// TIA Portal V16 export
// export: Created 2022-07-21T09:35:30.9300272Z, ExportSetting WithDefaults, DisplayName Totally Integrated Automation Portal, DisplayVersion V16 Update 4, DisplayName TIA Portal Version Control Interface, DisplayVersion V16 Update 2, DisplayName TIA Portal Openness, DisplayVersion V16 Update 4, DisplayName SINAMICS Startdrive Advanced, DisplayVersion V16 Update 5, DisplayName SINAMICS Startdrive G130, G150, S120, S150, SINAMICS MV, S210, DisplayVersion V16 Update 5, DisplayName SINAMICS Startdrive G110M, G120, G120C, G120D, G120P, G115D, DisplayVersion V16 Update 5, DisplayName STEP 7 Professional, DisplayVersion V16 Update 4, DisplayName STEP 7 Safety, DisplayVersion V16, DisplayName WinCC Advanced, DisplayVersion V16 Update 4
FUNCTION_BLOCK "fbTransport"   // FB34, LAD
TITLE = Transport handling / Obsługa transportu
{ S7_Optimized_Access := 'TRUE' }
VERSION : 0.1
// stored: AutoNumber true, IsIECCheckEnabled false, IsRetainMemResEnabled false, MemoryReserve 100, SetENOAutomatically false, UDAEnableTagReadback false
   VAR_INPUT
      inEnable { ExternalAccessible := 'False'; ExternalVisible := 'False'; ExternalWritable := 'False'} : Bool;   // Ogólne zezwolenie / General release
      inStartRelease { ExternalAccessible := 'False'; ExternalVisible := 'False'; ExternalWritable := 'False'} : Bool;   // Warunki na rozpoczęcie transportu / Conditions to start transport
      inLogOn { ExternalAccessible := 'False'; ExternalVisible := 'False'; ExternalWritable := 'False'} : Bool;   // Sygnał rozpoczynający transport / Start transport
      inLogOff { ExternalAccessible := 'False'; ExternalVisible := 'False'; ExternalWritable := 'False'} : Bool;   // Warunki na zakończenie transportu / Conditions to end transport
      inCancelTransport { ExternalAccessible := 'False'; ExternalVisible := 'False'; ExternalWritable := 'False'} : Bool;   // Natychmiastowe zakończenie transportu / Immediate end transport
      inNextPrevScan { ExternalAccessible := 'False'; ExternalVisible := 'False'; ExternalWritable := 'False'} : USInt;   // Dystans kolejnego przenośnika / Another conveyor distance
      inNextOnSpeed { ExternalAccessible := 'False'; ExternalVisible := 'False'; ExternalWritable := 'False'} : Bool;   // Następny przenośnik jedzie z nominalną prędkością / Next conveyor move with normal speed
      inHeadToHead { ExternalAccessible := 'False'; ExternalVisible := 'False'; ExternalWritable := 'False'} : UInt;   // Dystans czoło obiektu do czoła następnego / Distance head to next head
      inMinusToleranceHeadToHead { ExternalAccessible := 'False'; ExternalVisible := 'False'; ExternalWritable := 'False'} : UInt;   // Toleracja dystansu H2H / Distance tolerance H2H
      inTailToHead { ExternalAccessible := 'False'; ExternalVisible := 'False'; ExternalWritable := 'False'} : UInt;   // Dystans tył obiektu do następnego czoła / Distance tail to next head
      inMinusToleranceTailToHead { ExternalAccessible := 'False'; ExternalVisible := 'False'; ExternalWritable := 'False'} : UInt;   // Tolerancja dystansu T2H / Distance tolerance T2H
      inHeadToHeadTillCancel { ExternalAccessible := 'False'; ExternalVisible := 'False'; ExternalWritable := 'False'} : UInt := 0;   // Dystans do warunkowego zakończenia transportu / Distance to conditional end transport
   END_VAR
   VAR_IN_OUT
      ioData : "typeConveyor";   // Struktura conveyor / Conveyor structure
   END_VAR
   VAR
      sInternalEnable { ExternalAccessible := 'False'; ExternalVisible := 'False'; ExternalWritable := 'False'} : Bool;
   END_VAR
   VAR RETAIN
      sCounterHeadToHead { ExternalAccessible := 'False'; ExternalVisible := 'False'; ExternalWritable := 'False'} : UInt;
      sCounterTailToHead { ExternalAccessible := 'False'; ExternalVisible := 'False'; ExternalWritable := 'False'} : UInt;
      sCounterHeadToLogOn { ExternalAccessible := 'False'; ExternalVisible := 'False'; ExternalWritable := 'False'} : UInt;
      sMemRELogOn { ExternalAccessible := 'False'; ExternalVisible := 'False'; ExternalWritable := 'False'} : Bool;
      sMemRETransport { ExternalAccessible := 'False'; ExternalVisible := 'False'; ExternalWritable := 'False'} : Bool;
      sMemFETransport { ExternalAccessible := 'False'; ExternalVisible := 'False'; ExternalWritable := 'False'} : Bool;
   END_VAR
   VAR
      sHeadToHeadCancel : Bool;
   END_VAR
   VAR_TEMP
      tDistancePrevScan : USInt;
      tReqHeadToHead : UInt;
      tReqTailToHead : UInt;
      tTransportReady : Bool;
      tEndTransport : Bool;
      tDistanceReached : Bool;
      tReqMinusToleranceHeadToHead : UInt;
      tReqMinusToleranceTailToHead : UInt;
      tReset : Bool;
   END_VAR
   VAR_TEMP   // added for the SCL form of the ladder/FBD networks
      _w1 : Bool;
   END_VAR
BEGIN

REGION Network 1: Enable / Zezwolenie
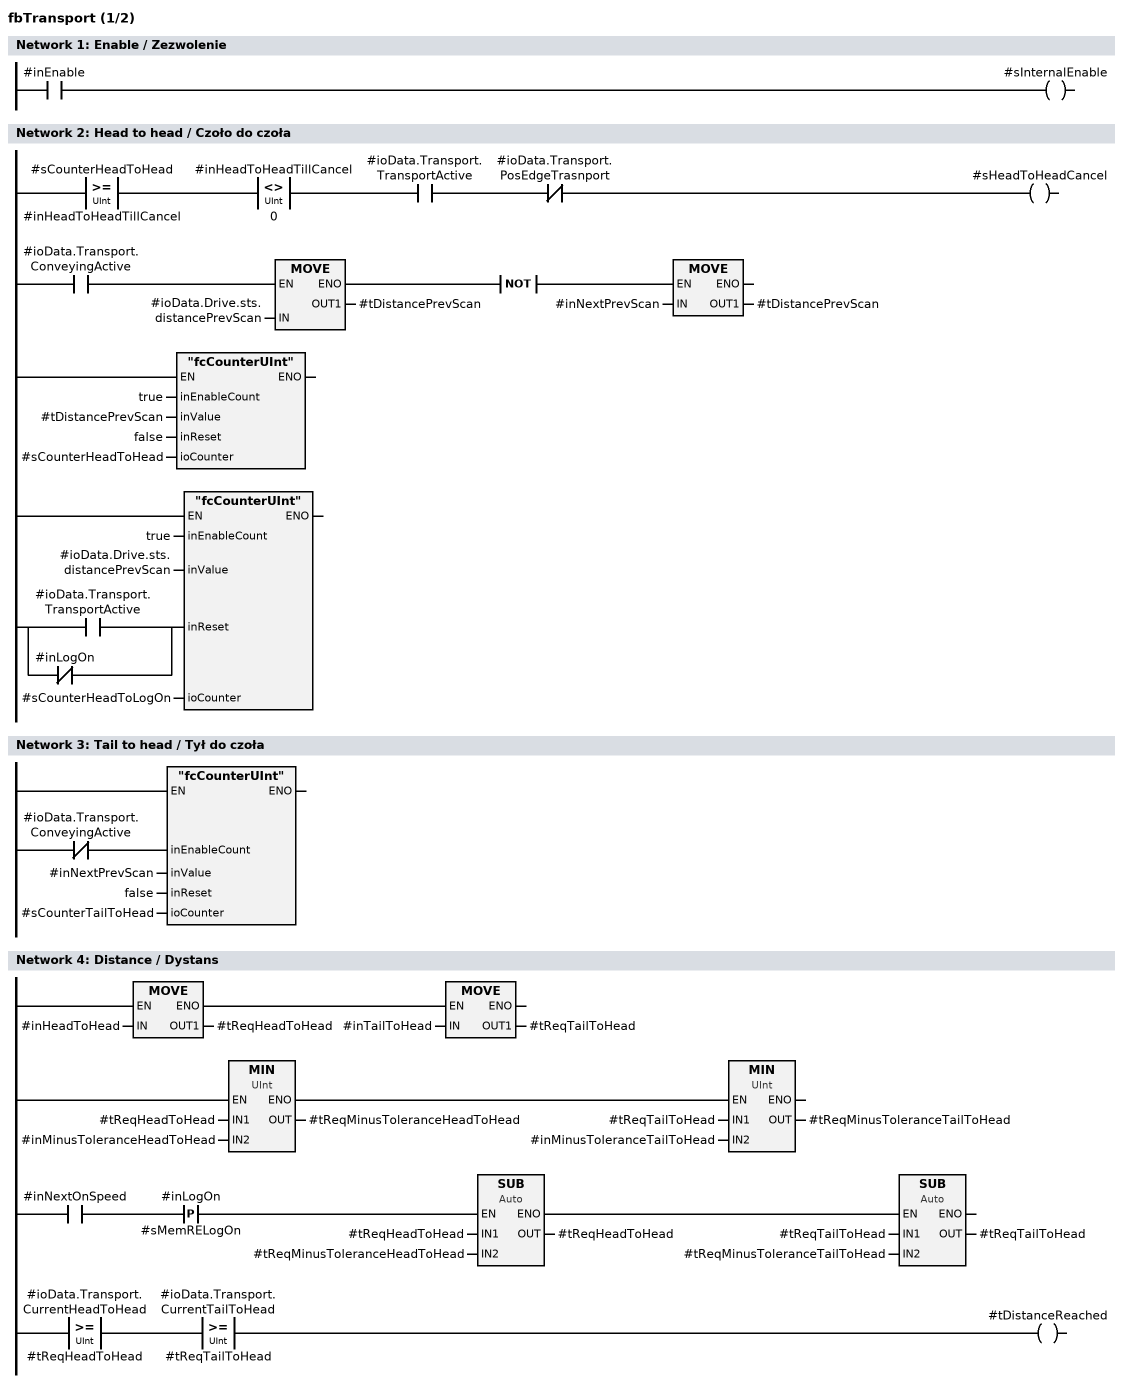
   RUNG wire#powerrail
      Contact( #inEnable )
      Coil( #sInternalEnable )
   END_RUNG
   // the same network as SCL:
   #sInternalEnable := #inEnable;
END_REGION

REGION Network 2: Head to head / Czoło do czoła
   RUNG wire#powerrail
      { S7_Templates := "SrcType := UInt" } GE_Contact(in1 := #sCounterHeadToHead, in2 := #inHeadToHeadTillCancel)
      { S7_Templates := "SrcType := UInt" } NE_Contact(in1 := #inHeadToHeadTillCancel, in2 := 0)
      Contact( #ioData.Transport.TransportActive )
      I_Contact( #ioData.Transport.PosEdgeTrasnport )
      Coil( #sHeadToHeadCancel )
   END_RUNG
   RUNG wire#powerrail
      Contact( #ioData.Transport.ConveyingActive )
      Move(in := #ioData.Drive.sts.distancePrevScan, out1 => #tDistancePrevScan)
      Not()
      Move(in := #inNextPrevScan, out1 => #tDistancePrevScan)
   END_RUNG
   RUNG wire#powerrail
      "fcCounterUInt"(inEnableCount := true, inValue := #tDistancePrevScan, inReset := false, ioCounter := #sCounterHeadToHead)
   END_RUNG
   RUNG wire#powerrail
      "fcCounterUInt"(inReset := wire#w1, inEnableCount := true, inValue := #ioData.Drive.sts.distancePrevScan, ioCounter := #sCounterHeadToLogOn)
   END_RUNG
   RUNG wire#powerrail
      Contact( #ioData.Transport.TransportActive )
   END_RUNG wire#w1
   RUNG wire#powerrail
      I_Contact( #inLogOn )
   END_RUNG wire#w1
   // the same network as SCL:
   #sHeadToHeadCancel := (#sCounterHeadToHead >= #inHeadToHeadTillCancel) AND (#inHeadToHeadTillCancel <> 0) AND #ioData.Transport.TransportActive AND NOT #ioData.Transport.PosEdgeTrasnport;
   IF #ioData.Transport.ConveyingActive THEN
       #tDistancePrevScan := #ioData.Drive.sts.distancePrevScan;
   END_IF;
   IF NOT #ioData.Transport.ConveyingActive THEN #tDistancePrevScan := #inNextPrevScan; END_IF;
   "fcCounterUInt"(inEnableCount := true,
                   inValue := #tDistancePrevScan,
                   inReset := false,
                   ioCounter := #sCounterHeadToHead);
   "fcCounterUInt"(inEnableCount := true,
                   inValue := #ioData.Drive.sts.distancePrevScan,
                   inReset := #ioData.Transport.TransportActive OR NOT #inLogOn,
                   ioCounter := #sCounterHeadToLogOn);
END_REGION

REGION Network 3: Tail to head / Tył do czoła
   RUNG wire#powerrail
      "fcCounterUInt"(inEnableCount := wire#w1, inValue := #inNextPrevScan, inReset := false, ioCounter := #sCounterTailToHead)
   END_RUNG
   RUNG wire#powerrail
      I_Contact( #ioData.Transport.ConveyingActive )
   END_RUNG wire#w1
   // the same network as SCL:
   "fcCounterUInt"(inEnableCount := NOT #ioData.Transport.ConveyingActive,
                   inValue := #inNextPrevScan,
                   inReset := false,
                   ioCounter := #sCounterTailToHead);
END_REGION

REGION Network 4: Distance / Dystans
   RUNG wire#powerrail
      Move(in := #inHeadToHead, out1 => #tReqHeadToHead)
      Move(in := #inTailToHead, out1 => #tReqTailToHead)
   END_RUNG
   RUNG wire#powerrail
      { S7_Templates := "[card := 2, value_type := UInt]" } MIN(in1 := #tReqHeadToHead, in2 := #inMinusToleranceHeadToHead, out => #tReqMinusToleranceHeadToHead)
      { S7_Templates := "[card := 2, value_type := UInt]" } MIN(in1 := #tReqTailToHead, in2 := #inMinusToleranceTailToHead, out => #tReqMinusToleranceTailToHead)
   END_RUNG
   RUNG wire#powerrail
      Contact( #inNextOnSpeed )
      P_Contact(operand := #inLogOn, bit := #sMemRELogOn)
      Sub(in1 := #tReqHeadToHead, in2 := #tReqMinusToleranceHeadToHead, out => #tReqHeadToHead)
      Sub(in1 := #tReqTailToHead, in2 := #tReqMinusToleranceTailToHead, out => #tReqTailToHead)
   END_RUNG
   RUNG wire#powerrail
      { S7_Templates := "SrcType := UInt" } GE_Contact(in1 := #ioData.Transport.CurrentHeadToHead, in2 := #tReqHeadToHead)
      { S7_Templates := "SrcType := UInt" } GE_Contact(in1 := #ioData.Transport.CurrentTailToHead, in2 := #tReqTailToHead)
      Coil( #tDistanceReached )
   END_RUNG
   // the same network as SCL:
   #tReqHeadToHead := #inHeadToHead;
   #tReqTailToHead := #inTailToHead;
   #tReqMinusToleranceHeadToHead := MIN(IN1 := #tReqHeadToHead, IN2 := #inMinusToleranceHeadToHead);
   #tReqMinusToleranceTailToHead := MIN(IN1 := #tReqTailToHead, IN2 := #inMinusToleranceTailToHead);
   #_w1 := #inNextOnSpeed AND #inLogOn AND NOT #sMemRELogOn;   // rising edge of #inLogOn
   #sMemRELogOn := #inLogOn;
   IF #_w1 THEN
       #tReqHeadToHead := #tReqHeadToHead - #tReqMinusToleranceHeadToHead;
       #tReqTailToHead := #tReqTailToHead - #tReqMinusToleranceTailToHead;
   END_IF;
   #tDistanceReached := (#ioData.Transport.CurrentHeadToHead >= #tReqHeadToHead) AND (#ioData.Transport.CurrentTailToHead >= #tReqTailToHead);
END_REGION

REGION Network 5: Transport
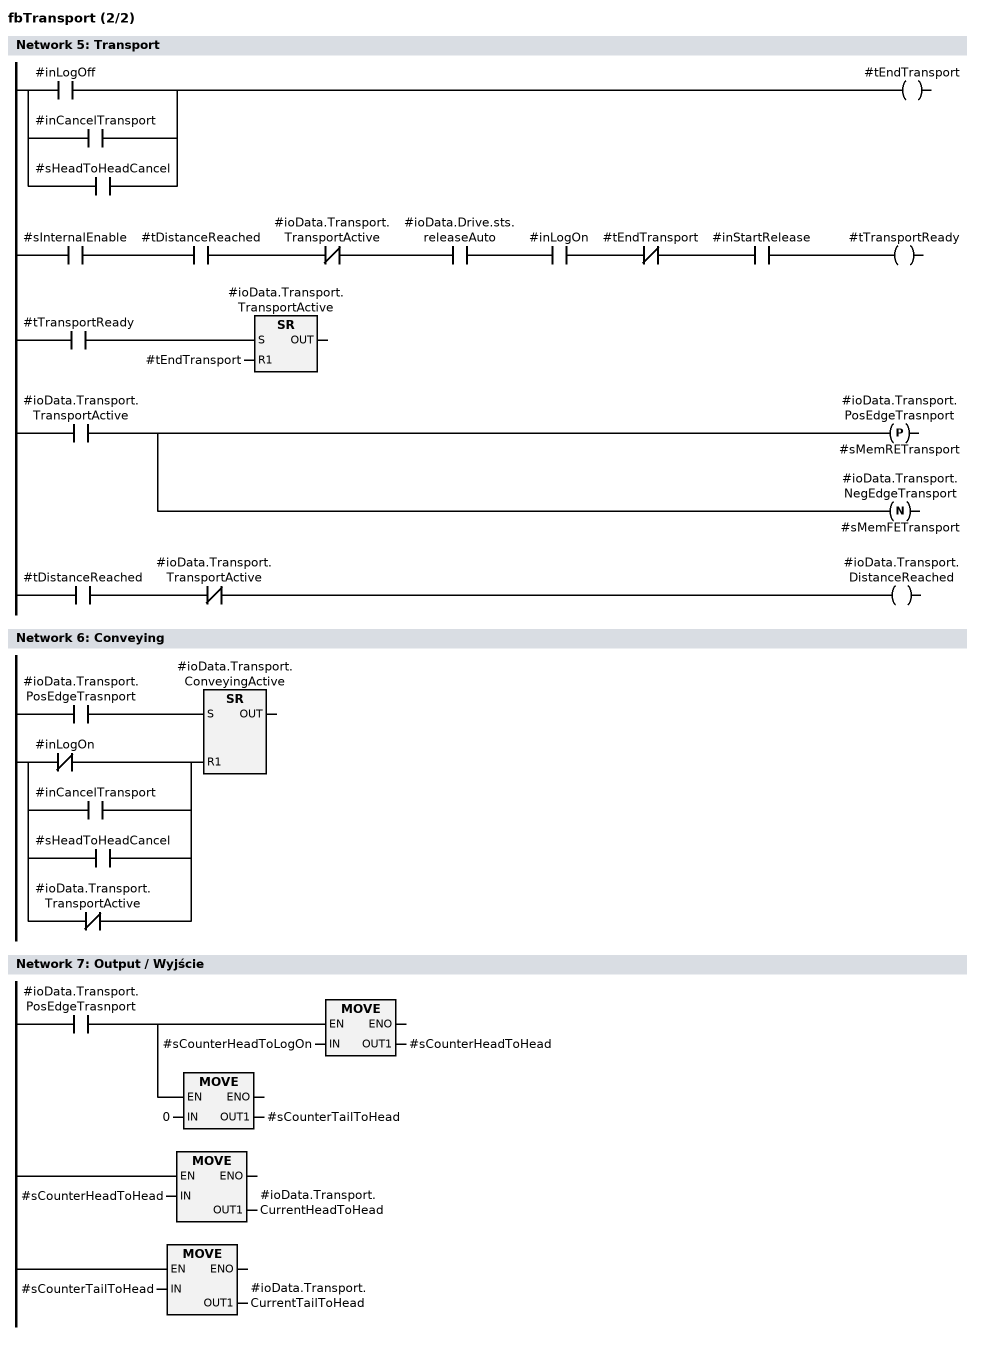
   #tEndTransport := #inLogOff OR #inCancelTransport OR #sHeadToHeadCancel;
   #tTransportReady := #sInternalEnable AND #tDistanceReached AND NOT #ioData.Transport.TransportActive AND #ioData.Drive.sts.releaseAuto AND #inLogOn AND NOT #tEndTransport AND #inStartRelease;
   IF #tTransportReady THEN
       #ioData.Transport.TransportActive := TRUE;   // SR flip-flop
   END_IF;
   IF #tEndTransport THEN #ioData.Transport.TransportActive := FALSE; END_IF;
   #ioData.Transport.PosEdgeTrasnport := #ioData.Transport.TransportActive AND NOT #sMemRETransport;   // rising edge
   #sMemRETransport := #ioData.Transport.TransportActive;
   #ioData.Transport.NegEdgeTransport := NOT #ioData.Transport.TransportActive AND #sMemFETransport;   // falling edge
   #sMemFETransport := #ioData.Transport.TransportActive;
   #ioData.Transport.DistanceReached := #tDistanceReached AND NOT #ioData.Transport.TransportActive;
END_REGION

REGION Network 6: Conveying
   RUNG wire#powerrail
      Contact( #ioData.Transport.PosEdgeTrasnport )
      S_SR(operand := #ioData.Transport.ConveyingActive, r1 := wire#w1)
   END_RUNG
   RUNG wire#powerrail
      I_Contact( #inLogOn )
   END_RUNG wire#w1
   RUNG wire#powerrail
      Contact( #inCancelTransport )
   END_RUNG wire#w1
   RUNG wire#powerrail
      Contact( #sHeadToHeadCancel )
   END_RUNG wire#w1
   RUNG wire#powerrail
      I_Contact( #ioData.Transport.TransportActive )
   END_RUNG wire#w1
   // the same network as SCL:
   IF #ioData.Transport.PosEdgeTrasnport THEN
       #ioData.Transport.ConveyingActive := TRUE;   // SR flip-flop
   END_IF;
   IF NOT #inLogOn OR #inCancelTransport OR #sHeadToHeadCancel OR NOT #ioData.Transport.TransportActive THEN
       #ioData.Transport.ConveyingActive := FALSE;
   END_IF;
END_REGION

REGION Network 7: Output / Wyjście
   RUNG wire#powerrail
      Contact( #ioData.Transport.PosEdgeTrasnport )
      wire#w1
      { S7_GenerateENO := "TRUE" } Move(in := #sCounterHeadToLogOn, out1 => #sCounterHeadToHead)
   END_RUNG
   RUNG wire#w1
      { S7_GenerateENO := "TRUE" } Move(in := 0, out1 => #sCounterTailToHead)
   END_RUNG
   RUNG wire#powerrail
      { S7_GenerateENO := "TRUE" } Move(in := #sCounterHeadToHead, out1 => #ioData.Transport.CurrentHeadToHead)
   END_RUNG
   RUNG wire#powerrail
      { S7_GenerateENO := "TRUE" } Move(in := #sCounterTailToHead, out1 => #ioData.Transport.CurrentTailToHead)
   END_RUNG
   // the same network as SCL:
   IF #ioData.Transport.PosEdgeTrasnport THEN
       #sCounterHeadToHead := #sCounterHeadToLogOn;
       #sCounterTailToHead := 0;
   END_IF;
   #ioData.Transport.CurrentHeadToHead := #sCounterHeadToHead;
   #ioData.Transport.CurrentTailToHead := #sCounterTailToHead;
END_REGION
END_FUNCTION_BLOCK
